{attribute 'qualified_only'}
{attribute 'strict'}
TYPE E_CX_State :
(
	IDLE,
	HW,
	OS,
	BASEFOLDER,
	DONE
);
END_TYPE

(* stored: Version 1.1.0.1
   DUT E_CX_State: Id {495df6fe-3219-40b3-b990-7bf5d5a3cc3b} *)
